   SPTP {A1 8.291, A2 -37.612, A3 70.753, A4 43.164, A5 -93.737, A6 0.000, E1 2824, E2 0, E3 0, E4 0, E5 0, E6 0} C_DIS
   SPTP {A1 8.655, A2 -38.617, A3 71.685, A4 45.116, A5 -92.691, A6 0.000, E1 2823.56, E2 0, E3 0, E4 0, E5 0, E6 0} C_DIS
   SPTP {A1 9.012, A2 -39.592, A3 72.518, A4 47.079, A5 -91.622, A6 0.000, E1 2823.06, E2 0, E3 0, E4 0, E5 0, E6 0} C_DIS
   SPTP {A1 9.360, A2 -40.537, A3 73.252, A4 49.063, A5 -90.537, A6 0.000, E1 2822.49, E2 0, E3 0, E4 0, E5 0, E6 0} C_DIS
   SPTP {A1 9.698, A2 -41.456, A3 73.903, A4 51.056, A5 -89.440, A6 0.000, E1 2821.87, E2 0, E3 0, E4 0, E5 0, E6 0} C_DIS
   SPTP {A1 10.024, A2 -42.359, A3 74.483, A4 53.057, A5 -88.326, A6 0.000, E1 2821.2, E2 0, E3 0, E4 0, E5 0, E6 0} C_DIS
   SPTP {A1 10.336, A2 -43.250, A3 75.008, A4 55.059, A5 -87.194, A6 0.000, E1 2820.49, E2 0, E3 0, E4 0, E5 0, E6 0} C_DIS
   SPTP {A1 10.632, A2 -44.132, A3 75.480, A4 57.062, A5 -86.046, A6 0.000, E1 2819.74, E2 0, E3 0, E4 0, E5 0, E6 0} C_DIS
   SPTP {A1 10.890, A2 -45.114, A3 76.113, A4 58.971, A5 -84.816, A6 0.000, E1 2818.78, E2 0, E3 0, E4 0, E5 0, E6 0} C_DIS
   SPTP {A1 11.121, A2 -46.138, A3 76.783, A4 60.845, A5 -83.533, A6 0.000, E1 2817.69, E2 0, E3 0, E4 0, E5 0, E6 0} C_DIS
   SPTP {A1 11.339, A2 -47.131, A3 77.364, A4 62.758, A5 -82.259, A6 0.000, E1 2816.52, E2 0, E3 0, E4 0, E5 0, E6 0} C_DIS
   SPTP {A1 11.539, A2 -48.119, A3 77.901, A4 64.680, A5 -80.965, A6 0.000, E1 2815.3, E2 0, E3 0, E4 0, E5 0, E6 0} C_DIS
   SPTP {A1 11.720, A2 -49.088, A3 78.371, A4 66.632, A5 -79.673, A6 0.000, E1 2814.01, E2 0, E3 0, E4 0, E5 0, E6 0} C_DIS
   SPTP {A1 11.880, A2 -50.051, A3 78.798, A4 68.601, A5 -78.370, A6 0.000, E1 2812.66, E2 0, E3 0, E4 0, E5 0, E6 0} C_DIS
   SPTP {A1 12.018, A2 -50.998, A3 79.170, A4 70.601, A5 -77.069, A6 0.000, E1 2811.24, E2 0, E3 0, E4 0, E5 0, E6 0} C_DIS
   SPTP {A1 12.134, A2 -51.928, A3 79.486, A4 72.635, A5 -75.777, A6 0.000, E1 2809.74, E2 0, E3 0, E4 0, E5 0, E6 0} C_DIS
   SPTP {A1 12.226, A2 -52.844, A3 79.754, A4 74.703, A5 -74.491, A6 0.000, E1 2808.16, E2 0, E3 0, E4 0, E5 0, E6 0} C_DIS
   SPTP {A1 12.294, A2 -53.734, A3 79.958, A4 76.821, A5 -73.233, A6 0.000, E1 2806.49, E2 0, E3 0, E4 0, E5 0, E6 0} C_DIS
   SPTP {A1 12.336, A2 -54.611, A3 80.117, A4 78.978, A5 -71.988, A6 0.000, E1 2804.74, E2 0, E3 0, E4 0, E5 0, E6 0} C_DIS
   SPTP {A1 12.353, A2 -55.450, A3 80.202, A4 81.200, A5 -70.792, A6 0.000, E1 2802.89, E2 0, E3 0, E4 0, E5 0, E6 0} C_DIS
   SPTP {A1 12.342, A2 -56.273, A3 80.242, A4 83.468, A5 -69.622, A6 0.000, E1 2800.95, E2 0, E3 0, E4 0, E5 0, E6 0} C_DIS
   SPTP {A1 12.305, A2 -57.043, A3 80.209, A4 85.765, A5 -68.529, A6 0.000, E1 2798.98, E2 0, E3 0, E4 0, E5 0, E6 0} C_DIS
   SPTP {A1 12.237, A2 -57.731, A3 80.168, A4 87.843, A5 -67.518, A6 0.000, E1 2797.48, E2 0, E3 0, E4 0, E5 0, E6 0} C_DIS
   SPTP {A1 12.145, A2 -58.394, A3 80.097, A4 89.941, A5 -66.542, A6 0.000, E1 2795.96, E2 0, E3 0, E4 0, E5 0, E6 0} C_DIS
   SPTP {A1 12.029, A2 -59.039, A3 79.995, A4 92.086, A5 -65.598, A6 0.000, E1 2794.37, E2 0, E3 0, E4 0, E5 0, E6 0} C_DIS
   SPTP {A1 11.888, A2 -59.661, A3 79.859, A4 94.281, A5 -64.695, A6 0.000, E1 2792.7, E2 0, E3 0, E4 0, E5 0, E6 0} C_DIS
   SPTP {A1 11.725, A2 -60.257, A3 79.681, A4 96.532, A5 -63.846, A6 0.000, E1 2790.95, E2 0, E3 0, E4 0, E5 0, E6 0} C_DIS
   SPTP {A1 11.538, A2 -60.826, A3 79.463, A4 98.838, A5 -63.054, A6 0.000, E1 2789.12, E2 0, E3 0, E4 0, E5 0, E6 0} C_DIS
   SPTP {A1 11.330, A2 -61.356, A3 79.191, A4 101.205, A5 -62.342, A6 0.000, E1 2787.21, E2 0, E3 0, E4 0, E5 0, E6 0} C_DIS
   SPTP {A1 11.102, A2 -61.846, A3 78.877, A4 103.596, A5 -61.710, A6 0.000, E1 2785.3, E2 0, E3 0, E4 0, E5 0, E6 0} C_DIS
   SPTP {A1 10.857, A2 -62.345, A3 78.828, A4 105.431, A5 -60.901, A6 0.000, E1 2784.47, E2 0, E3 0, E4 0, E5 0, E6 0} C_DIS
   SPTP {A1 10.594, A2 -62.833, A3 78.769, A4 107.306, A5 -60.114, A6 0.000, E1 2783.59, E2 0, E3 0, E4 0, E5 0, E6 0} C_DIS
   SPTP {A1 10.316, A2 -63.305, A3 78.697, A4 109.222, A5 -59.358, A6 0.000, E1 2782.66, E2 0, E3 0, E4 0, E5 0, E6 0} C_DIS
   SPTP {A1 10.023, A2 -63.754, A3 78.603, A4 111.183, A5 -58.650, A6 0.000, E1 2781.69, E2 0, E3 0, E4 0, E5 0, E6 0} C_DIS
   SPTP {A1 9.720, A2 -64.176, A3 78.479, A4 113.187, A5 -58.005, A6 0.000, E1 2780.67, E2 0, E3 0, E4 0, E5 0, E6 0} C_DIS
   SPTP {A1 9.408, A2 -64.567, A3 78.320, A4 115.233, A5 -57.433, A6 0.000, E1 2779.62, E2 0, E3 0, E4 0, E5 0, E6 0} C_DIS
   SPTP {A1 9.091, A2 -65.008, A3 78.418, A4 116.875, A5 -56.634, A6 0.000, E1 2779.28, E2 0, E3 0, E4 0, E5 0, E6 0} C_DIS
   SPTP {A1 8.770, A2 -65.530, A3 78.839, A4 118.046, A5 -55.511, A6 0.000, E1 2779.72, E2 0, E3 0, E4 0, E5 0, E6 0} C_DIS
   SPTP {A1 8.446, A2 -66.037, A3 79.254, A4 119.230, A5 -54.404, A6 0.000, E1 2780.16, E2 0, E3 0, E4 0, E5 0, E6 0} C_DIS
   SPTP {A1 8.121, A2 -66.525, A3 79.661, A4 120.426, A5 -53.321, A6 0.000, E1 2780.59, E2 0, E3 0, E4 0, E5 0, E6 0} C_DIS
   SPTP {A1 7.799, A2 -66.994, A3 80.058, A4 121.629, A5 -52.270, A6 0.000, E1 2781.03, E2 0, E3 0, E4 0, E5 0, E6 0} C_DIS
   SPTP {A1 7.483, A2 -67.468, A3 80.529, A4 122.693, A5 -51.156, A6 0.000, E1 2781.68, E2 0, E3 0, E4 0, E5 0, E6 0} C_DIS
   SPTP {A1 7.179, A2 -68.121, A3 81.695, A4 122.558, A5 -49.253, A6 0.000, E1 2784.01, E2 0, E3 0, E4 0, E5 0, E6 0} C_DIS
   SPTP {A1 6.881, A2 -68.742, A3 82.846, A4 122.311, A5 -47.360, A6 0.000, E1 2786.45, E2 0, E3 0, E4 0, E5 0, E6 0} C_DIS
   SPTP {A1 6.594, A2 -69.329, A3 83.978, A4 121.941, A5 -45.490, A6 0.000, E1 2788.99, E2 0, E3 0, E4 0, E5 0, E6 0} C_DIS
   SPTP {A1 6.318, A2 -69.881, A3 85.088, A4 121.431, A5 -43.647, A6 0.000, E1 2791.66, E2 0, E3 0, E4 0, E5 0, E6 0} C_DIS
   SPTP {A1 6.056, A2 -70.415, A3 86.267, A4 120.536, A5 -41.738, A6 0.000, E1 2794.76, E2 0, E3 0, E4 0, E5 0, E6 0} C_DIS
   SPTP {A1 5.815, A2 -71.014, A3 88.060, A4 117.608, A5 -39.163, A6 0.000, E1 2800.21, E2 0, E3 0, E4 0, E5 0, E6 0} C_DIS
   SPTP {A1 5.586, A2 -71.518, A3 89.769, A4 114.120, A5 -36.768, A6 0.000, E1 2806.19, E2 0, E3 0, E4 0, E5 0, E6 0} C_DIS
   SPTP {A1 5.369, A2 -71.925, A3 91.391, A4 110.015, A5 -34.596, A6 0.000, E1 2812.75, E2 0, E3 0, E4 0, E5 0, E6 0} C_DIS
   SPTP {A1 5.164, A2 -72.236, A3 92.924, A4 105.256, A5 -32.692, A6 0.000, E1 2819.92, E2 0, E3 0, E4 0, E5 0, E6 0} C_DIS
   SPTP {A1 4.973, A2 -72.448, A3 94.361, A4 99.843, A5 -31.125, A6 0.000, E1 2827.73, E2 0, E3 0, E4 0, E5 0, E6 0} C_DIS
   SPTP {A1 4.799, A2 -72.541, A3 95.781, A4 93.294, A5 -29.981, A6 0.000, E1 2836.62, E2 0, E3 0, E4 0, E5 0, E6 0} C_DIS
   SPTP {A1 4.634, A2 -72.488, A3 97.196, A4 85.489, A5 -29.420, A6 0.000, E1 2846.72, E2 0, E3 0, E4 0, E5 0, E6 0} C_DIS
   SPTP {A1 4.476, A2 -72.304, A3 98.465, A4 77.540, A5 -29.493, A6 0.000, E1 2856.93, E2 0, E3 0, E4 0, E5 0, E6 0} C_DIS
   SPTP {A1 4.325, A2 -71.991, A3 99.585, A4 69.822, A5 -30.191, A6 0.000, E1 2866.89, E2 0, E3 0, E4 0, E5 0, E6 0} C_DIS
   SPTP {A1 4.184, A2 -71.551, A3 100.551, A4 62.659, A5 -31.470, A6 0.000, E1 2876.29, E2 0, E3 0, E4 0, E5 0, E6 0} C_DIS
   SPTP {A1 4.057, A2 -70.984, A3 101.355, A4 56.273, A5 -33.255, A6 0.000, E1 2884.92, E2 0, E3 0, E4 0, E5 0, E6 0} C_DIS
   SPTP {A1 3.945, A2 -70.297, A3 101.995, A4 50.740, A5 -35.451, A6 0.000, E1 2892.7, E2 0, E3 0, E4 0, E5 0, E6 0} C_DIS
   SPTP {A1 3.847, A2 -69.498, A3 102.471, A4 46.033, A5 -37.961, A6 0.000, E1 2899.67, E2 0, E3 0, E4 0, E5 0, E6 0} C_DIS
   SPTP {A1 3.765, A2 -68.591, A3 102.779, A4 42.097, A5 -40.706, A6 0.000, E1 2905.88, E2 0, E3 0, E4 0, E5 0, E6 0} C_DIS
   SPTP {A1 3.703, A2 -67.583, A3 102.917, A4 38.849, A5 -43.620, A6 0.000, E1 2911.44, E2 0, E3 0, E4 0, E5 0, E6 0} C_DIS
   SPTP {A1 3.653, A2 -66.854, A3 102.974, A4 36.807, A5 -45.736, A6 0.000, E1 2915.49, E2 0, E3 0, E4 0, E5 0, E6 0} C_DIS
   SPTP {A1 3.624, A2 -66.078, A3 102.937, A4 35.090, A5 -47.900, A6 0.000, E1 2919.25, E2 0, E3 0, E4 0, E5 0, E6 0} C_DIS
   SPTP {A1 3.613, A2 -65.259, A3 102.808, A4 33.656, A5 -50.096, A6 0.000, E1 2922.75, E2 0, E3 0, E4 0, E5 0, E6 0} C_DIS
   SPTP {A1 3.621, A2 -64.401, A3 102.588, A4 32.476, A5 -52.305, A6 0.000, E1 2926.04, E2 0, E3 0, E4 0, E5 0, E6 0} C_DIS
   SPTP {A1 3.649, A2 -63.505, A3 102.276, A4 31.531, A5 -54.518, A6 0.000, E1 2929.12, E2 0, E3 0, E4 0, E5 0, E6 0} C_DIS
   SPTP {A1 3.697, A2 -62.577, A3 101.874, A4 30.798, A5 -56.719, A6 0.000, E1 2932.04, E2 0, E3 0, E4 0, E5 0, E6 0} C_DIS
   SPTP {A1 3.784, A2 -61.839, A3 101.495, A4 30.469, A5 -58.436, A6 0.000, E1 2934.56, E2 0, E3 0, E4 0, E5 0, E6 0} C_DIS
   SPTP {A1 3.910, A2 -61.333, A3 101.190, A4 30.506, A5 -59.622, A6 0.000, E1 2936.71, E2 0, E3 0, E4 0, E5 0, E6 0} C_DIS
   SPTP {A1 4.054, A2 -60.816, A3 100.844, A4 30.653, A5 -60.796, A6 0.000, E1 2938.79, E2 0, E3 0, E4 0, E5 0, E6 0} C_DIS
   SPTP {A1 4.213, A2 -60.292, A3 100.460, A4 30.895, A5 -61.956, A6 0.000, E1 2940.8, E2 0, E3 0, E4 0, E5 0, E6 0} C_DIS
   SPTP {A1 4.383, A2 -59.761, A3 100.041, A4 31.211, A5 -63.096, A6 0.000, E1 2942.75, E2 0, E3 0, E4 0, E5 0, E6 0} C_DIS
   SPTP {A1 4.563, A2 -59.225, A3 99.586, A4 31.603, A5 -64.215, A6 0.000, E1 2944.66, E2 0, E3 0, E4 0, E5 0, E6 0} C_DIS
   SPTP {A1 4.753, A2 -58.683, A3 99.094, A4 32.066, A5 -65.312, A6 0.000, E1 2946.51, E2 0, E3 0, E4 0, E5 0, E6 0} C_DIS
   SPTP {A1 4.951, A2 -58.137, A3 98.569, A4 32.587, A5 -66.385, A6 0.000, E1 2948.32, E2 0, E3 0, E4 0, E5 0, E6 0} C_DIS
   SPTP {A1 5.200, A2 -57.839, A3 98.169, A4 33.422, A5 -66.957, A6 0.000, E1 2949.88, E2 0, E3 0, E4 0, E5 0, E6 0} C_DIS
   SPTP {A1 5.478, A2 -57.668, A3 97.826, A4 34.439, A5 -67.271, A6 0.000, E1 2951.28, E2 0, E3 0, E4 0, E5 0, E6 0} C_DIS
   SPTP {A1 5.759, A2 -57.494, A3 97.460, A4 35.497, A5 -67.574, A6 0.000, E1 2952.65, E2 0, E3 0, E4 0, E5 0, E6 0} C_DIS
   SPTP {A1 6.043, A2 -57.319, A3 97.070, A4 36.589, A5 -67.865, A6 0.000, E1 2953.99, E2 0, E3 0, E4 0, E5 0, E6 0} C_DIS
   SPTP {A1 6.327, A2 -57.140, A3 96.658, A4 37.712, A5 -68.146, A6 0.000, E1 2955.29, E2 0, E3 0, E4 0, E5 0, E6 0} C_DIS
   SPTP {A1 6.613, A2 -56.959, A3 96.222, A4 38.865, A5 -68.416, A6 0.000, E1 2956.57, E2 0, E3 0, E4 0, E5 0, E6 0} C_DIS
   SPTP {A1 6.896, A2 -56.775, A3 95.765, A4 40.039, A5 -68.676, A6 0.000, E1 2957.82, E2 0, E3 0, E4 0, E5 0, E6 0} C_DIS
   SPTP {A1 7.178, A2 -56.589, A3 95.287, A4 41.232, A5 -68.926, A6 0.000, E1 2959.05, E2 0, E3 0, E4 0, E5 0, E6 0} C_DIS
   SPTP {A1 7.456, A2 -56.402, A3 94.790, A4 42.440, A5 -69.166, A6 0.000, E1 2960.26, E2 0, E3 0, E4 0, E5 0, E6 0} C_DIS
   SPTP {A1 7.729, A2 -56.213, A3 94.273, A4 43.658, A5 -69.394, A6 0.000, E1 2961.45, E2 0, E3 0, E4 0, E5 0, E6 0} C_DIS
   SPTP {A1 7.996, A2 -56.024, A3 93.742, A4 44.880, A5 -69.610, A6 0.000, E1 2962.63, E2 0, E3 0, E4 0, E5 0, E6 0} C_DIS
   SPTP {A1 8.257, A2 -55.836, A3 93.196, A4 46.105, A5 -69.815, A6 0.000, E1 2963.81, E2 0, E3 0, E4 0, E5 0, E6 0} C_DIS
   SPTP {A1 8.523, A2 -55.760, A3 92.717, A4 47.443, A5 -69.822, A6 0.000, E1 2964.79, E2 0, E3 0, E4 0, E5 0, E6 0} C_DIS
   SPTP {A1 8.783, A2 -55.694, A3 92.230, A4 48.797, A5 -69.805, A6 0.000, E1 2965.75, E2 0, E3 0, E4 0, E5 0, E6 0} C_DIS
   SPTP {A1 9.034, A2 -55.626, A3 91.728, A4 50.152, A5 -69.783, A6 0.000, E1 2966.69, E2 0, E3 0, E4 0, E5 0, E6 0} C_DIS
   SPTP {A1 9.278, A2 -55.557, A3 91.213, A4 51.506, A5 -69.757, A6 0.000, E1 2967.63, E2 0, E3 0, E4 0, E5 0, E6 0} C_DIS
   SPTP {A1 9.512, A2 -55.488, A3 90.688, A4 52.857, A5 -69.725, A6 0.000, E1 2968.55, E2 0, E3 0, E4 0, E5 0, E6 0} C_DIS
   SPTP {A1 9.737, A2 -55.420, A3 90.153, A4 54.202, A5 -69.688, A6 0.000, E1 2969.47, E2 0, E3 0, E4 0, E5 0, E6 0} C_DIS
   SPTP {A1 9.953, A2 -55.353, A3 89.611, A4 55.538, A5 -69.645, A6 0.000, E1 2970.39, E2 0, E3 0, E4 0, E5 0, E6 0} C_DIS
   SPTP {A1 10.158, A2 -55.289, A3 89.065, A4 56.865, A5 -69.594, A6 0.000, E1 2971.3, E2 0, E3 0, E4 0, E5 0, E6 0} C_DIS
   SPTP {A1 10.352, A2 -55.227, A3 88.515, A4 58.180, A5 -69.536, A6 0.000, E1 2972.22, E2 0, E3 0, E4 0, E5 0, E6 0} C_DIS
   SPTP {A1 10.536, A2 -55.171, A3 87.966, A4 59.481, A5 -69.468, A6 0.000, E1 2973.14, E2 0, E3 0, E4 0, E5 0, E6 0} C_DIS
   SPTP {A1 10.700, A2 -55.122, A3 87.442, A4 60.719, A5 -69.407, A6 0.000, E1 2974.04, E2 0, E3 0, E4 0, E5 0, E6 0} C_DIS
   SPTP {A1 10.850, A2 -55.080, A3 86.931, A4 61.923, A5 -69.341, A6 0.000, E1 2974.94, E2 0, E3 0, E4 0, E5 0, E6 0} C_DIS
   SPTP {A1 10.965, A2 -55.046, A3 86.490, A4 62.972, A5 -69.312, A6 0.000, E1 2975.8, E2 0, E3 0, E4 0, E5 0, E6 0} C_DIS
   SPTP {A1 11.068, A2 -55.022, A3 86.067, A4 63.988, A5 -69.273, A6 0.000, E1 2976.66, E2 0, E3 0, E4 0, E5 0, E6 0} C_DIS
   SPTP {A1 11.164, A2 -55.008, A3 85.655, A4 64.986, A5 -69.221, A6 0.000, E1 2977.54, E2 0, E3 0, E4 0, E5 0, E6 0} C_DIS
   SPTP {A1 11.250, A2 -55.004, A3 85.258, A4 65.965, A5 -69.153, A6 0.000, E1 2978.43, E2 0, E3 0, E4 0, E5 0, E6 0} C_DIS
   SPTP {A1 11.329, A2 -55.012, A3 84.876, A4 66.925, A5 -69.067, A6 0.000, E1 2979.34, E2 0, E3 0, E4 0, E5 0, E6 0} C_DIS
   SPTP {A1 11.400, A2 -55.031, A3 84.511, A4 67.865, A5 -68.964, A6 0.000, E1 2980.26, E2 0, E3 0, E4 0, E5 0, E6 0} C_DIS
   SPTP {A1 11.462, A2 -55.065, A3 84.166, A4 68.784, A5 -68.840, A6 0.000, E1 2981.19, E2 0, E3 0, E4 0, E5 0, E6 0} C_DIS
   SPTP {A1 11.516, A2 -55.112, A3 83.842, A4 69.683, A5 -68.696, A6 0.000, E1 2982.14, E2 0, E3 0, E4 0, E5 0, E6 0} C_DIS
   SPTP {A1 11.562, A2 -55.174, A3 83.539, A4 70.561, A5 -68.529, A6 0.000, E1 2983.1, E2 0, E3 0, E4 0, E5 0, E6 0} C_DIS
   SPTP {A1 11.600, A2 -55.251, A3 83.260, A4 71.418, A5 -68.340, A6 0.000, E1 2984.08, E2 0, E3 0, E4 0, E5 0, E6 0} C_DIS
   SPTP {A1 11.630, A2 -55.344, A3 83.006, A4 72.254, A5 -68.126, A6 0.000, E1 2985.08, E2 0, E3 0, E4 0, E5 0, E6 0} C_DIS
   SPTP {A1 11.652, A2 -55.453, A3 82.777, A4 73.069, A5 -67.888, A6 0.000, E1 2986.09, E2 0, E3 0, E4 0, E5 0, E6 0} C_DIS
   SPTP {A1 11.666, A2 -55.579, A3 82.575, A4 73.863, A5 -67.625, A6 0.000, E1 2987.12, E2 0, E3 0, E4 0, E5 0, E6 0} C_DIS
   SPTP {A1 11.672, A2 -55.721, A3 82.401, A4 74.635, A5 -67.334, A6 0.000, E1 2988.17, E2 0, E3 0, E4 0, E5 0, E6 0} C_DIS
   SPTP {A1 11.671, A2 -55.881, A3 82.255, A4 75.387, A5 -67.016, A6 0.000, E1 2989.23, E2 0, E3 0, E4 0, E5 0, E6 0} C_DIS
   SPTP {A1 11.661, A2 -56.058, A3 82.138, A4 76.117, A5 -66.670, A6 0.000, E1 2990.3, E2 0, E3 0, E4 0, E5 0, E6 0} C_DIS
   SPTP {A1 11.644, A2 -56.253, A3 82.050, A4 76.826, A5 -66.293, A6 0.000, E1 2991.4, E2 0, E3 0, E4 0, E5 0, E6 0} C_DIS
   SPTP {A1 11.611, A2 -56.512, A3 82.046, A4 77.547, A5 -65.858, A6 0.000, E1 2992.22, E2 0, E3 0, E4 0, E5 0, E6 0} C_DIS
   SPTP {A1 11.571, A2 -56.791, A3 82.070, A4 78.258, A5 -65.397, A6 0.000, E1 2993.02, E2 0, E3 0, E4 0, E5 0, E6 0} C_DIS
   SPTP {A1 11.523, A2 -57.080, A3 82.113, A4 78.957, A5 -64.914, A6 0.000, E1 2993.82, E2 0, E3 0, E4 0, E5 0, E6 0} C_DIS
   SPTP {A1 11.468, A2 -57.383, A3 82.178, A4 79.641, A5 -64.406, A6 0.000, E1 2994.62, E2 0, E3 0, E4 0, E5 0, E6 0} C_DIS
   SPTP {A1 11.406, A2 -57.697, A3 82.264, A4 80.312, A5 -63.873, A6 0.000, E1 2995.44, E2 0, E3 0, E4 0, E5 0, E6 0} C_DIS
   SPTP {A1 11.336, A2 -58.025, A3 82.371, A4 80.968, A5 -63.314, A6 0.000, E1 2996.26, E2 0, E3 0, E4 0, E5 0, E6 0} C_DIS
   SPTP {A1 11.258, A2 -58.365, A3 82.500, A4 81.609, A5 -62.728, A6 0.000, E1 2997.08, E2 0, E3 0, E4 0, E5 0, E6 0} C_DIS
   SPTP {A1 11.173, A2 -58.718, A3 82.651, A4 82.236, A5 -62.114, A6 0.000, E1 2997.91, E2 0, E3 0, E4 0, E5 0, E6 0} C_DIS
   SPTP {A1 11.079, A2 -59.083, A3 82.823, A4 82.849, A5 -61.473, A6 0.000, E1 2998.75, E2 0, E3 0, E4 0, E5 0, E6 0} C_DIS
   SPTP {A1 10.977, A2 -59.459, A3 83.015, A4 83.448, A5 -60.804, A6 0.000, E1 2999.59, E2 0, E3 0, E4 0, E5 0, E6 0} C_DIS
   SPTP {A1 10.867, A2 -59.846, A3 83.228, A4 84.033, A5 -60.106, A6 0.000, E1 3000.43, E2 0, E3 0, E4 0, E5 0, E6 0} C_DIS
   SPTP {A1 10.748, A2 -60.245, A3 83.460, A4 84.605, A5 -59.379, A6 0.000, E1 3001.28, E2 0, E3 0, E4 0, E5 0, E6 0} C_DIS
   SPTP {A1 10.629, A2 -60.717, A3 83.597, A4 85.698, A5 -58.495, A6 0.000, E1 3001.52, E2 0, E3 0, E4 0, E5 0, E6 0} C_DIS
   SPTP {A1 10.498, A2 -61.191, A3 83.738, A4 86.804, A5 -57.596, A6 0.000, E1 3001.74, E2 0, E3 0, E4 0, E5 0, E6 0} C_DIS
   SPTP {A1 10.355, A2 -61.668, A3 83.884, A4 87.922, A5 -56.684, A6 0.000, E1 3001.94, E2 0, E3 0, E4 0, E5 0, E6 0} C_DIS
   SPTP {A1 10.201, A2 -62.146, A3 84.036, A4 89.054, A5 -55.758, A6 0.000, E1 3002.1, E2 0, E3 0, E4 0, E5 0, E6 0} C_DIS
   SPTP {A1 10.036, A2 -62.624, A3 84.192, A4 90.203, A5 -54.820, A6 0.000, E1 3002.24, E2 0, E3 0, E4 0, E5 0, E6 0} C_DIS
   SPTP {A1 9.859, A2 -63.102, A3 84.351, A4 91.371, A5 -53.873, A6 0.000, E1 3002.35, E2 0, E3 0, E4 0, E5 0, E6 0} C_DIS
   SPTP {A1 9.670, A2 -63.579, A3 84.513, A4 92.559, A5 -52.914, A6 0.000, E1 3002.42, E2 0, E3 0, E4 0, E5 0, E6 0} C_DIS
   SPTP {A1 9.469, A2 -64.055, A3 84.678, A4 93.770, A5 -51.944, A6 0.000, E1 3002.46, E2 0, E3 0, E4 0, E5 0, E6 0} C_DIS
   SPTP {A1 9.257, A2 -64.531, A3 84.846, A4 95.006, A5 -50.964, A6 0.000, E1 3002.46, E2 0, E3 0, E4 0, E5 0, E6 0} C_DIS
   SPTP {A1 9.032, A2 -65.004, A3 85.017, A4 96.271, A5 -49.974, A6 0.000, E1 3002.43, E2 0, E3 0, E4 0, E5 0, E6 0} C_DIS
   SPTP {A1 8.795, A2 -65.475, A3 85.190, A4 97.566, A5 -48.977, A6 0.000, E1 3002.34, E2 0, E3 0, E4 0, E5 0, E6 0} C_DIS
   SPTP {A1 8.545, A2 -65.943, A3 85.363, A4 98.896, A5 -47.972, A6 0.000, E1 3002.22, E2 0, E3 0, E4 0, E5 0, E6 0} C_DIS
   SPTP {A1 8.284, A2 -66.407, A3 85.538, A4 100.264, A5 -46.962, A6 0.000, E1 3002.04, E2 0, E3 0, E4 0, E5 0, E6 0} C_DIS
   SPTP {A1 8.011, A2 -66.866, A3 85.711, A4 101.674, A5 -45.950, A6 0.000, E1 3001.81, E2 0, E3 0, E4 0, E5 0, E6 0} C_DIS
   SPTP {A1 7.724, A2 -67.320, A3 85.859, A4 103.228, A5 -44.926, A6 0.000, E1 3001.47, E2 0, E3 0, E4 0, E5 0, E6 0} C_DIS
   SPTP {A1 7.411, A2 -67.777, A3 85.920, A4 105.216, A5 -43.841, A6 0.000, E1 3000.88, E2 0, E3 0, E4 0, E5 0, E6 0} C_DIS
   SPTP {A1 7.084, A2 -68.223, A3 85.976, A4 107.281, A5 -42.777, A6 0.000, E1 3000.19, E2 0, E3 0, E4 0, E5 0, E6 0} C_DIS
   SPTP {A1 6.742, A2 -68.658, A3 86.030, A4 109.428, A5 -41.733, A6 0.000, E1 2999.42, E2 0, E3 0, E4 0, E5 0, E6 0} C_DIS
   SPTP {A1 6.386, A2 -69.081, A3 86.080, A4 111.660, A5 -40.713, A6 0.000, E1 2998.55, E2 0, E3 0, E4 0, E5 0, E6 0} C_DIS
   SPTP {A1 6.016, A2 -69.492, A3 86.128, A4 113.983, A5 -39.720, A6 0.000, E1 2997.59, E2 0, E3 0, E4 0, E5 0, E6 0} C_DIS
   SPTP {A1 5.634, A2 -69.889, A3 86.169, A4 116.400, A5 -38.763, A6 0.000, E1 2996.52, E2 0, E3 0, E4 0, E5 0, E6 0} C_DIS
   SPTP {A1 5.240, A2 -70.272, A3 86.205, A4 118.913, A5 -37.851, A6 0.000, E1 2995.36, E2 0, E3 0, E4 0, E5 0, E6 0} C_DIS
   SPTP {A1 4.837, A2 -70.638, A3 86.234, A4 121.523, A5 -36.988, A6 0.000, E1 2994.11, E2 0, E3 0, E4 0, E5 0, E6 0} C_DIS
   SPTP {A1 4.425, A2 -70.989, A3 86.256, A4 124.227, A5 -36.181, A6 0.000, E1 2992.76, E2 0, E3 0, E4 0, E5 0, E6 0} C_DIS
   SPTP {A1 4.006, A2 -71.322, A3 86.271, A4 127.019, A5 -35.437, A6 0.000, E1 2991.32, E2 0, E3 0, E4 0, E5 0, E6 0} C_DIS
   SPTP {A1 3.581, A2 -71.639, A3 86.281, A4 129.897, A5 -34.756, A6 0.000, E1 2989.81, E2 0, E3 0, E4 0, E5 0, E6 0} C_DIS
   SPTP {A1 3.149, A2 -71.941, A3 86.286, A4 132.852, A5 -34.141, A6 0.000, E1 2988.23, E2 0, E3 0, E4 0, E5 0, E6 0} C_DIS
   SPTP {A1 2.715, A2 -72.225, A3 86.284, A4 135.865, A5 -33.605, A6 0.000, E1 2986.6, E2 0, E3 0, E4 0, E5 0, E6 0} C_DIS
   SPTP {A1 2.281, A2 -72.555, A3 86.514, A4 138.429, A5 -32.773, A6 0.000, E1 2985.54, E2 0, E3 0, E4 0, E5 0, E6 0} C_DIS
   SPTP {A1 1.845, A2 -72.929, A3 86.959, A4 140.623, A5 -31.635, A6 0.000, E1 2984.96, E2 0, E3 0, E4 0, E5 0, E6 0} C_DIS
   SPTP {A1 1.413, A2 -73.291, A3 87.411, A4 142.897, A5 -30.522, A6 0.000, E1 2984.3, E2 0, E3 0, E4 0, E5 0, E6 0} C_DIS
   SPTP {A1 0.983, A2 -73.642, A3 87.869, A4 145.255, A5 -29.433, A6 0.000, E1 2983.56, E2 0, E3 0, E4 0, E5 0, E6 0} C_DIS
   SPTP {A1 0.564, A2 -73.981, A3 88.333, A4 147.674, A5 -28.380, A6 0.000, E1 2982.77, E2 0, E3 0, E4 0, E5 0, E6 0} C_DIS
   SPTP {A1 0.158, A2 -74.307, A3 88.803, A4 150.140, A5 -27.366, A6 0.000, E1 2981.96, E2 0, E3 0, E4 0, E5 0, E6 0} C_DIS
   SPTP {A1 -0.229, A2 -74.622, A3 89.278, A4 152.627, A5 -26.396, A6 0.000, E1 2981.14, E2 0, E3 0, E4 0, E5 0, E6 0} C_DIS
   SPTP {A1 -0.592, A2 -74.973, A3 89.961, A4 154.675, A5 -25.088, A6 0.000, E1 2980.8, E2 0, E3 0, E4 0, E5 0, E6 0} C_DIS
   SPTP {A1 -0.921, A2 -75.415, A3 91.154, A4 155.531, A5 -22.825, A6 0.000, E1 2981.64, E2 0, E3 0, E4 0, E5 0, E6 0} C_DIS
   SPTP {A1 -1.221, A2 -75.822, A3 92.330, A4 156.269, A5 -20.565, A6 0.000, E1 2982.62, E2 0, E3 0, E4 0, E5 0, E6 0} C_DIS
   SPTP {A1 -1.484, A2 -76.194, A3 93.486, A4 156.798, A5 -18.315, A6 0.000, E1 2983.83, E2 0, E3 0, E4 0, E5 0, E6 0} C_DIS
   SPTP {A1 -1.707, A2 -76.530, A3 94.623, A4 156.983, A5 -16.077, A6 0.000, E1 2985.4, E2 0, E3 0, E4 0, E5 0, E6 0} C_DIS
   SPTP {A1 -1.878, A2 -76.847, A3 95.938, A4 155.655, A5 -13.412, A6 0.000, E1 2988.51, E2 0, E3 0, E4 0, E5 0, E6 0} C_DIS
   SPTP {A1 -2.003, A2 -77.121, A3 97.769, A4 148.572, A5 -9.513, A6 0.000, E1 2997.32, E2 0, E3 0, E4 0, E5 0, E6 0} C_DIS
   SPTP {A1 -2.073, A2 -77.268, A3 99.483, A4 131.076, A5 -6.066, A6 0.000, E1 3016.55, E2 0, E3 0, E4 0, E5 0, E6 0} C_DIS
   SPTP {A1 -2.095, A2 -77.287, A3 101.076, A4 87.723, A5 -4.353, A6 0.000, E1 3061.65, E2 0, E3 0, E4 0, E5 0, E6 0} C_DIS
   SPTP {A1 -2.058, A2 -77.175, A3 102.538, A4 44.883, A5 -6.134, A6 0.000, E1 3106.26, E2 0, E3 0, E4 0, E5 0, E6 0} C_DIS
   SPTP {A1 -1.985, A2 -76.714, A3 104.288, A4 23.426, A5 -11.222, A6 0.000, E1 3129.5, E2 0, E3 0, E4 0, E5 0, E6 0} C_DIS
   SPTP {A1 -1.870, A2 -75.910, A3 105.843, A4 15.959, A5 -17.402, A6 0.000, E1 3138.75, E2 0, E3 0, E4 0, E5 0, E6 0} C_DIS
   SPTP {A1 -1.718, A2 -74.815, A3 107.046, A4 12.881, A5 -23.708, A6 0.000, E1 3143.62, E2 0, E3 0, E4 0, E5 0, E6 0} C_DIS
   SPTP {A1 -1.548, A2 -73.241, A3 107.939, A4 11.064, A5 -30.738, A6 0.000, E1 3147.32, E2 0, E3 0, E4 0, E5 0, E6 0} C_DIS
   SPTP {A1 -1.356, A2 -70.901, A3 108.348, A4 9.830, A5 -39.024, A6 0.000, E1 3150.66, E2 0, E3 0, E4 0, E5 0, E6 0} C_DIS
   SPTP {A1 -1.158, A2 -68.174, A3 108.071, A4 9.263, A5 -47.048, A6 0.000, E1 3153.34, E2 0, E3 0, E4 0, E5 0, E6 0} C_DIS
   SPTP {A1 -0.962, A2 -65.135, A3 107.107, A4 9.065, A5 -54.717, A6 0.000, E1 3155.68, E2 0, E3 0, E4 0, E5 0, E6 0} C_DIS
   SPTP {A1 -0.727, A2 -62.038, A3 105.570, A4 9.217, A5 -61.595, A6 0.000, E1 3157.91, E2 0, E3 0, E4 0, E5 0, E6 0} C_DIS
   SPTP {A1 -0.305, A2 -59.408, A3 103.857, A4 10.064, A5 -66.874, A6 0.000, E1 3160.23, E2 0, E3 0, E4 0, E5 0, E6 0} C_DIS
   SPTP {A1 0.131, A2 -56.724, A3 101.755, A4 11.050, A5 -71.795, A6 0.000, E1 3162.51, E2 0, E3 0, E4 0, E5 0, E6 0} C_DIS
   SPTP {A1 0.584, A2 -54.011, A3 99.275, A4 12.190, A5 -76.346, A6 0.000, E1 3164.75, E2 0, E3 0, E4 0, E5 0, E6 0} C_DIS
   SPTP {A1 1.046, A2 -51.291, A3 96.439, A4 13.453, A5 -80.520, A6 0.000, E1 3166.97, E2 0, E3 0, E4 0, E5 0, E6 0} C_DIS
   SPTP {A1 1.511, A2 -48.578, A3 93.262, A4 14.831, A5 -84.315, A6 0.000, E1 3169.17, E2 0, E3 0, E4 0, E5 0, E6 0} C_DIS
   SPTP {A1 1.980, A2 -45.874, A3 89.752, A4 16.327, A5 -87.740, A6 0.000, E1 3171.33, E2 0, E3 0, E4 0, E5 0, E6 0} C_DIS
   SPTP {A1 2.453, A2 -43.174, A3 85.904, A4 17.952, A5 -90.804, A6 0.000, E1 3173.44, E2 0, E3 0, E4 0, E5 0, E6 0} C_DIS
   SPTP {A1 2.923, A2 -40.469, A3 81.717, A4 19.679, A5 -93.514, A6 0.000, E1 3175.49, E2 0, E3 0, E4 0, E5 0, E6 0} C_DIS
   SPTP {A1 3.388, A2 -37.736, A3 77.160, A4 21.509, A5 -95.879, A6 0.000, E1 3177.44, E2 0, E3 0, E4 0, E5 0, E6 0} C_DIS
   SPTP {A1 3.843, A2 -34.945, A3 72.200, A4 23.417, A5 -97.903, A6 0.000, E1 3179.27, E2 0, E3 0, E4 0, E5 0, E6 0} C_DIS
   SPTP {A1 4.407, A2 -34.766, A3 71.380, A4 25.593, A5 -97.876, A6 0.000, E1 3180.54, E2 0, E3 0, E4 0, E5 0, E6 0} C_DIS
   SPTP {A1 4.967, A2 -34.634, A3 70.580, A4 27.841, A5 -97.769, A6 0.000, E1 3181.65, E2 0, E3 0, E4 0, E5 0, E6 0} C_DIS
   SPTP {A1 5.517, A2 -34.477, A3 69.685, A4 30.139, A5 -97.636, A6 0.000, E1 3182.61, E2 0, E3 0, E4 0, E5 0, E6 0} C_DIS
   SPTP {A1 6.038, A2 -34.559, A3 69.172, A4 32.400, A5 -97.327, A6 0.000, E1 3183.34, E2 0, E3 0, E4 0, E5 0, E6 0} C_DIS
   SPTP {A1 6.516, A2 -35.196, A3 69.605, A4 34.539, A5 -96.655, A6 0.000, E1 3183.71, E2 0, E3 0, E4 0, E5 0, E6 0} C_DIS
   SPTP {A1 6.983, A2 -35.782, A3 69.912, A4 36.702, A5 -95.978, A6 0.000, E1 3183.95, E2 0, E3 0, E4 0, E5 0, E6 0} C_DIS
   SPTP {A1 7.440, A2 -36.329, A3 70.111, A4 38.888, A5 -95.294, A6 0.000, E1 3184.09, E2 0, E3 0, E4 0, E5 0, E6 0} C_DIS
   SPTP {A1 7.441, A2 -36.315, A3 70.093, A4 38.902, A5 -95.305, A6 0.000, E1 3184.07, E2 0, E3 0, E4 0, E5 0, E6 0} C_DIS
   SPTP {A1 7.888, A2 -36.831, A3 70.201, A4 41.107, A5 -94.614, A6 0.000, E1 3184.15, E2 0, E3 0, E4 0, E5 0, E6 0} C_DIS
   SPTP {A1 8.292, A2 -37.590, A3 70.724, A4 43.181, A5 -93.755, A6 0.000, E1 3183.98, E2 0, E3 0, E4 0, E5 0, E6 0} C_DIS
   SPTP {A1 8.656, A2 -38.593, A3 71.652, A4 45.135, A5 -92.711, A6 0.000, E1 3183.53, E2 0, E3 0, E4 0, E5 0, E6 0} C_DIS
   SPTP {A1 9.013, A2 -39.567, A3 72.483, A4 47.099, A5 -91.644, A6 0.000, E1 3183.03, E2 0, E3 0, E4 0, E5 0, E6 0} C_DIS
   SPTP {A1 9.362, A2 -40.510, A3 73.216, A4 49.084, A5 -90.562, A6 0.000, E1 3182.46, E2 0, E3 0, E4 0, E5 0, E6 0} C_DIS
   SPTP {A1 9.700, A2 -41.428, A3 73.864, A4 51.078, A5 -89.467, A6 0.000, E1 3181.83, E2 0, E3 0, E4 0, E5 0, E6 0} C_DIS
   SPTP {A1 10.026, A2 -42.329, A3 74.443, A4 53.080, A5 -88.355, A6 0.000, E1 3181.17, E2 0, E3 0, E4 0, E5 0, E6 0} C_DIS
   SPTP {A1 10.338, A2 -43.220, A3 74.967, A4 55.082, A5 -87.225, A6 0.000, E1 3180.46, E2 0, E3 0, E4 0, E5 0, E6 0} C_DIS
   SPTP {A1 10.634, A2 -44.100, A3 75.438, A4 57.085, A5 -86.079, A6 0.000, E1 3179.71, E2 0, E3 0, E4 0, E5 0, E6 0} C_DIS
   SPTP {A1 10.892, A2 -45.082, A3 76.070, A4 58.995, A5 -84.852, A6 0.000, E1 3178.75, E2 0, E3 0, E4 0, E5 0, E6 0} C_DIS
   SPTP {A1 11.124, A2 -46.105, A3 76.740, A4 60.870, A5 -83.571, A6 0.000, E1 3177.66, E2 0, E3 0, E4 0, E5 0, E6 0} C_DIS
   SPTP {A1 11.342, A2 -47.097, A3 77.320, A4 62.782, A5 -82.299, A6 0.000, E1 3176.49, E2 0, E3 0, E4 0, E5 0, E6 0} C_DIS
   SPTP {A1 11.542, A2 -48.085, A3 77.857, A4 64.705, A5 -81.006, A6 0.000, E1 3175.27, E2 0, E3 0, E4 0, E5 0, E6 0} C_DIS
   SPTP {A1 11.723, A2 -49.054, A3 78.327, A4 66.656, A5 -79.716, A6 0.000, E1 3173.98, E2 0, E3 0, E4 0, E5 0, E6 0} C_DIS
   SPTP {A1 11.883, A2 -50.016, A3 78.755, A4 68.625, A5 -78.414, A6 0.000, E1 3172.64, E2 0, E3 0, E4 0, E5 0, E6 0} C_DIS
   SPTP {A1 12.022, A2 -50.963, A3 79.127, A4 70.624, A5 -77.116, A6 0.000, E1 3171.21, E2 0, E3 0, E4 0, E5 0, E6 0} C_DIS
   SPTP {A1 12.139, A2 -51.893, A3 79.444, A4 72.657, A5 -75.825, A6 0.000, E1 3169.72, E2 0, E3 0, E4 0, E5 0, E6 0} C_DIS
   SPTP {A1 12.231, A2 -52.810, A3 79.713, A4 74.725, A5 -74.540, A6 0.000, E1 3168.14, E2 0, E3 0, E4 0, E5 0, E6 0} C_DIS
   SPTP {A1 12.299, A2 -53.700, A3 79.917, A4 76.841, A5 -73.283, A6 0.000, E1 3166.48, E2 0, E3 0, E4 0, E5 0, E6 0} C_DIS
   SPTP {A1 12.341, A2 -54.576, A3 80.078, A4 78.997, A5 -72.039, A6 0.000, E1 3164.73, E2 0, E3 0, E4 0, E5 0, E6 0} C_DIS
   SPTP {A1 12.359, A2 -55.416, A3 80.163, A4 81.217, A5 -70.844, A6 0.000, E1 3162.88, E2 0, E3 0, E4 0, E5 0, E6 0} C_DIS
   SPTP {A1 12.348, A2 -56.240, A3 80.205, A4 83.484, A5 -69.674, A6 0.000, E1 3160.94, E2 0, E3 0, E4 0, E5 0, E6 0} C_DIS
   SPTP {A1 12.311, A2 -57.011, A3 80.174, A4 85.778, A5 -68.581, A6 0.000, E1 3158.98, E2 0, E3 0, E4 0, E5 0, E6 0} C_DIS
   SPTP {A1 12.243, A2 -57.699, A3 80.134, A4 87.855, A5 -67.569, A6 0.000, E1 3157.48, E2 0, E3 0, E4 0, E5 0, E6 0} C_DIS
   SPTP {A1 12.152, A2 -58.363, A3 80.065, A4 89.951, A5 -66.593, A6 0.000, E1 3155.96, E2 0, E3 0, E4 0, E5 0, E6 0} C_DIS
   SPTP {A1 12.036, A2 -59.009, A3 79.965, A4 92.092, A5 -65.648, A6 0.000, E1 3154.38, E2 0, E3 0, E4 0, E5 0, E6 0} C_DIS
   SPTP {A1 11.896, A2 -59.633, A3 79.830, A4 94.285, A5 -64.745, A6 0.000, E1 3152.71, E2 0, E3 0, E4 0, E5 0, E6 0} C_DIS
   SPTP {A1 11.732, A2 -60.230, A3 79.655, A4 96.533, A5 -63.895, A6 0.000, E1 3150.96, E2 0, E3 0, E4 0, E5 0, E6 0} C_DIS
   SPTP {A1 11.545, A2 -60.799, A3 79.440, A4 98.835, A5 -63.101, A6 0.000, E1 3149.14, E2 0, E3 0, E4 0, E5 0, E6 0} C_DIS
   SPTP {A1 11.337, A2 -61.331, A3 79.170, A4 101.199, A5 -62.386, A6 0.000, E1 3147.23, E2 0, E3 0, E4 0, E5 0, E6 0} C_DIS
   SPTP {A1 11.110, A2 -61.823, A3 78.857, A4 103.591, A5 -61.753, A6 0.000, E1 3145.31, E2 0, E3 0, E4 0, E5 0, E6 0} C_DIS
   SPTP {A1 10.864, A2 -62.323, A3 78.810, A4 105.423, A5 -60.942, A6 0.000, E1 3144.49, E2 0, E3 0, E4 0, E5 0, E6 0} C_DIS
   SPTP {A1 10.602, A2 -62.812, A3 78.754, A4 107.295, A5 -60.152, A6 0.000, E1 3143.61, E2 0, E3 0, E4 0, E5 0, E6 0} C_DIS
   SPTP {A1 10.323, A2 -63.286, A3 78.685, A4 109.208, A5 -59.393, A6 0.000, E1 3142.69, E2 0, E3 0, E4 0, E5 0, E6 0} C_DIS
   SPTP {A1 10.031, A2 -63.737, A3 78.593, A4 111.166, A5 -58.682, A6 0.000, E1 3141.71, E2 0, E3 0, E4 0, E5 0, E6 0} C_DIS
   SPTP {A1 9.728, A2 -64.161, A3 78.471, A4 113.167, A5 -58.034, A6 0.000, E1 3140.7, E2 0, E3 0, E4 0, E5 0, E6 0} C_DIS
   SPTP {A1 9.416, A2 -64.553, A3 78.315, A4 115.210, A5 -57.458, A6 0.000, E1 3139.65, E2 0, E3 0, E4 0, E5 0, E6 0} C_DIS
   SPTP {A1 9.098, A2 -64.995, A3 78.410, A4 116.859, A5 -56.662, A6 0.000, E1 3139.29, E2 0, E3 0, E4 0, E5 0, E6 0} C_DIS
   SPTP {A1 8.776, A2 -65.518, A3 78.833, A4 118.029, A5 -55.534, A6 0.000, E1 3139.73, E2 0, E3 0, E4 0, E5 0, E6 0} C_DIS
   SPTP {A1 8.452, A2 -66.026, A3 79.251, A4 119.211, A5 -54.423, A6 0.000, E1 3140.17, E2 0, E3 0, E4 0, E5 0, E6 0} C_DIS
   SPTP {A1 8.126, A2 -66.517, A3 79.661, A4 120.405, A5 -53.336, A6 0.000, E1 3140.6, E2 0, E3 0, E4 0, E5 0, E6 0} C_DIS
   SPTP {A1 7.804, A2 -66.987, A3 80.059, A4 121.607, A5 -52.282, A6 0.000, E1 3141.03, E2 0, E3 0, E4 0, E5 0, E6 0} C_DIS
   SPTP {A1 7.487, A2 -67.459, A3 80.522, A4 122.689, A5 -51.177, A6 0.000, E1 3141.65, E2 0, E3 0, E4 0, E5 0, E6 0} C_DIS
   SPTP {A1 7.182, A2 -68.113, A3 81.688, A4 122.555, A5 -49.272, A6 0.000, E1 3143.98, E2 0, E3 0, E4 0, E5 0, E6 0} C_DIS
   SPTP {A1 6.884, A2 -68.736, A3 82.840, A4 122.312, A5 -47.376, A6 0.000, E1 3146.41, E2 0, E3 0, E4 0, E5 0, E6 0} C_DIS
   SPTP {A1 6.595, A2 -69.324, A3 83.972, A4 121.944, A5 -45.503, A6 0.000, E1 3148.94, E2 0, E3 0, E4 0, E5 0, E6 0} C_DIS
   SPTP {A1 6.318, A2 -69.877, A3 85.083, A4 121.439, A5 -43.658, A6 0.000, E1 3151.61, E2 0, E3 0, E4 0, E5 0, E6 0} C_DIS
   SPTP {A1 6.055, A2 -70.409, A3 86.248, A4 120.584, A5 -41.762, A6 0.000, E1 3154.65, E2 0, E3 0, E4 0, E5 0, E6 0} C_DIS
   SPTP {A1 5.812, A2 -71.010, A3 88.042, A4 117.670, A5 -39.183, A6 0.000, E1 3160.09, E2 0, E3 0, E4 0, E5 0, E6 0} C_DIS
   SPTP {A1 5.583, A2 -71.516, A3 89.750, A4 114.197, A5 -36.784, A6 0.000, E1 3166.05, E2 0, E3 0, E4 0, E5 0, E6 0} C_DIS
   SPTP {A1 5.365, A2 -71.925, A3 91.372, A4 110.109, A5 -34.606, A6 0.000, E1 3172.59, E2 0, E3 0, E4 0, E5 0, E6 0} C_DIS
   SPTP {A1 5.159, A2 -72.238, A3 92.906, A4 105.366, A5 -32.694, A6 0.000, E1 3179.74, E2 0, E3 0, E4 0, E5 0, E6 0} C_DIS
   SPTP {A1 4.966, A2 -72.452, A3 94.345, A4 99.967, A5 -31.116, A6 0.000, E1 3187.52, E2 0, E3 0, E4 0, E5 0, E6 0} C_DIS
   SPTP {A1 4.792, A2 -72.549, A3 95.759, A4 93.468, A5 -29.960, A6 0.000, E1 3196.37, E2 0, E3 0, E4 0, E5 0, E6 0} C_DIS
   SPTP {A1 4.626, A2 -72.500, A3 97.176, A4 85.670, A5 -29.383, A6 0.000, E1 3206.45, E2 0, E3 0, E4 0, E5 0, E6 0} C_DIS
   SPTP {A1 4.467, A2 -72.320, A3 98.448, A4 77.717, A5 -29.438, A6 0.000, E1 3216.67, E2 0, E3 0, E4 0, E5 0, E6 0} C_DIS
   SPTP {A1 4.316, A2 -72.011, A3 99.571, A4 69.987, A5 -30.121, A6 0.000, E1 3226.64, E2 0, E3 0, E4 0, E5 0, E6 0} C_DIS
   SPTP {A1 4.174, A2 -71.575, A3 100.540, A4 62.804, A5 -31.383, A6 0.000, E1 3236.06, E2 0, E3 0, E4 0, E5 0, E6 0} C_DIS
   SPTP {A1 4.048, A2 -71.012, A3 101.347, A4 56.397, A5 -33.156, A6 0.000, E1 3244.7, E2 0, E3 0, E4 0, E5 0, E6 0} C_DIS
   SPTP {A1 3.935, A2 -70.330, A3 101.992, A4 50.843, A5 -35.340, A6 0.000, E1 3252.5, E2 0, E3 0, E4 0, E5 0, E6 0} C_DIS
   SPTP {A1 3.837, A2 -69.535, A3 102.473, A4 46.116, A5 -37.841, A6 0.000, E1 3259.49, E2 0, E3 0, E4 0, E5 0, E6 0} C_DIS
   SPTP {A1 3.756, A2 -68.632, A3 102.786, A4 42.165, A5 -40.580, A6 0.000, E1 3265.71, E2 0, E3 0, E4 0, E5 0, E6 0} C_DIS
   SPTP {A1 3.694, A2 -67.629, A3 102.929, A4 38.902, A5 -43.488, A6 0.000, E1 3271.28, E2 0, E3 0, E4 0, E5 0, E6 0} C_DIS
   SPTP {A1 3.644, A2 -66.888, A3 102.987, A4 36.825, A5 -45.637, A6 0.000, E1 3275.38, E2 0, E3 0, E4 0, E5 0, E6 0} C_DIS
   SPTP {A1 3.615, A2 -66.115, A3 102.953, A4 35.102, A5 -47.799, A6 0.000, E1 3279.14, E2 0, E3 0, E4 0, E5 0, E6 0} C_DIS
   SPTP {A1 3.604, A2 -65.298, A3 102.828, A4 33.663, A5 -49.993, A6 0.000, E1 3282.65, E2 0, E3 0, E4 0, E5 0, E6 0} C_DIS
   SPTP {A1 3.612, A2 -64.441, A3 102.611, A4 32.479, A5 -52.202, A6 0.000, E1 3285.93, E2 0, E3 0, E4 0, E5 0, E6 0} C_DIS
   SPTP {A1 3.641, A2 -63.548, A3 102.303, A4 31.532, A5 -54.414, A6 0.000, E1 3289.02, E2 0, E3 0, E4 0, E5 0, E6 0} C_DIS
   SPTP {A1 3.688, A2 -62.621, A3 101.904, A4 30.796, A5 -56.615, A6 0.000, E1 3291.93, E2 0, E3 0, E4 0, E5 0, E6 0} C_DIS
   SPTP {A1 3.773, A2 -61.863, A3 101.517, A4 30.443, A5 -58.378, A6 0.000, E1 3294.48, E2 0, E3 0, E4 0, E5 0, E6 0} C_DIS
   SPTP {A1 3.899, A2 -61.357, A3 101.214, A4 30.478, A5 -59.564, A6 0.000, E1 3296.63, E2 0, E3 0, E4 0, E5 0, E6 0} C_DIS
   SPTP {A1 4.044, A2 -60.841, A3 100.869, A4 30.625, A5 -60.740, A6 0.000, E1 3298.71, E2 0, E3 0, E4 0, E5 0, E6 0} C_DIS
   SPTP {A1 4.202, A2 -60.317, A3 100.486, A4 30.866, A5 -61.900, A6 0.000, E1 3300.71, E2 0, E3 0, E4 0, E5 0, E6 0} C_DIS
   SPTP {A1 4.372, A2 -59.786, A3 100.069, A4 31.181, A5 -63.040, A6 0.000, E1 3302.67, E2 0, E3 0, E4 0, E5 0, E6 0} C_DIS
   SPTP {A1 4.552, A2 -59.250, A3 99.615, A4 31.573, A5 -64.160, A6 0.000, E1 3304.57, E2 0, E3 0, E4 0, E5 0, E6 0} C_DIS
   SPTP {A1 4.742, A2 -58.709, A3 99.125, A4 32.033, A5 -65.258, A6 0.000, E1 3306.42, E2 0, E3 0, E4 0, E5 0, E6 0} C_DIS
   SPTP {A1 4.939, A2 -58.163, A3 98.602, A4 32.552, A5 -66.332, A6 0.000, E1 3308.23, E2 0, E3 0, E4 0, E5 0, E6 0} C_DIS
   SPTP {A1 5.185, A2 -57.844, A3 98.190, A4 33.366, A5 -66.945, A6 0.000, E1 3309.81, E2 0, E3 0, E4 0, E5 0, E6 0} C_DIS
   SPTP {A1 5.462, A2 -57.673, A3 97.848, A4 34.381, A5 -67.260, A6 0.000, E1 3311.21, E2 0, E3 0, E4 0, E5 0, E6 0} C_DIS
   SPTP {A1 5.744, A2 -57.499, A3 97.482, A4 35.438, A5 -67.564, A6 0.000, E1 3312.58, E2 0, E3 0, E4 0, E5 0, E6 0} C_DIS
   SPTP {A1 6.027, A2 -57.324, A3 97.094, A4 36.528, A5 -67.856, A6 0.000, E1 3313.91, E2 0, E3 0, E4 0, E5 0, E6 0} C_DIS
   SPTP {A1 6.312, A2 -57.145, A3 96.683, A4 37.650, A5 -68.137, A6 0.000, E1 3315.22, E2 0, E3 0, E4 0, E5 0, E6 0} C_DIS
   SPTP {A1 6.597, A2 -56.964, A3 96.249, A4 38.801, A5 -68.408, A6 0.000, E1 3316.49, E2 0, E3 0, E4 0, E5 0, E6 0} C_DIS
   SPTP {A1 6.881, A2 -56.780, A3 95.793, A4 39.974, A5 -68.669, A6 0.000, E1 3317.74, E2 0, E3 0, E4 0, E5 0, E6 0} C_DIS
   SPTP {A1 7.162, A2 -56.594, A3 95.316, A4 41.166, A5 -68.920, A6 0.000, E1 3318.97, E2 0, E3 0, E4 0, E5 0, E6 0} C_DIS
   SPTP {A1 7.440, A2 -56.406, A3 94.819, A4 42.373, A5 -69.160, A6 0.000, E1 3320.18, E2 0, E3 0, E4 0, E5 0, E6 0} C_DIS
   SPTP {A1 7.714, A2 -56.217, A3 94.304, A4 43.590, A5 -69.390, A6 0.000, E1 3321.37, E2 0, E3 0, E4 0, E5 0, E6 0} C_DIS
   SPTP {A1 7.981, A2 -56.029, A3 93.774, A4 44.811, A5 -69.607, A6 0.000, E1 3322.56, E2 0, E3 0, E4 0, E5 0, E6 0} C_DIS
   SPTP {A1 8.243, A2 -55.841, A3 93.229, A4 46.035, A5 -69.812, A6 0.000, E1 3323.73, E2 0, E3 0, E4 0, E5 0, E6 0} C_DIS
   SPTP {A1 8.508, A2 -55.757, A3 92.745, A4 47.364, A5 -69.833, A6 0.000, E1 3324.73, E2 0, E3 0, E4 0, E5 0, E6 0} C_DIS
   SPTP {A1 8.768, A2 -55.691, A3 92.259, A4 48.716, A5 -69.816, A6 0.000, E1 3325.68, E2 0, E3 0, E4 0, E5 0, E6 0} C_DIS
   SPTP {A1 9.020, A2 -55.623, A3 91.759, A4 50.070, A5 -69.795, A6 0.000, E1 3326.63, E2 0, E3 0, E4 0, E5 0, E6 0} C_DIS
   SPTP {A1 9.263, A2 -55.554, A3 91.245, A4 51.423, A5 -69.769, A6 0.000, E1 3327.56, E2 0, E3 0, E4 0, E5 0, E6 0} C_DIS
   SPTP {A1 9.498, A2 -55.485, A3 90.721, A4 52.772, A5 -69.738, A6 0.000, E1 3328.49, E2 0, E3 0, E4 0, E5 0, E6 0} C_DIS
   SPTP {A1 9.724, A2 -55.417, A3 90.187, A4 54.116, A5 -69.701, A6 0.000, E1 3329.41, E2 0, E3 0, E4 0, E5 0, E6 0} C_DIS
   SPTP {A1 9.939, A2 -55.350, A3 89.646, A4 55.452, A5 -69.658, A6 0.000, E1 3330.32, E2 0, E3 0, E4 0, E5 0, E6 0} C_DIS
   SPTP {A1 10.145, A2 -55.285, A3 89.100, A4 56.778, A5 -69.607, A6 0.000, E1 3331.24, E2 0, E3 0, E4 0, E5 0, E6 0} C_DIS
   SPTP {A1 10.340, A2 -55.224, A3 88.551, A4 58.093, A5 -69.551, A6 0.000, E1 3332.15, E2 0, E3 0, E4 0, E5 0, E6 0} C_DIS
   SPTP {A1 10.525, A2 -55.168, A3 88.002, A4 59.393, A5 -69.483, A6 0.000, E1 3333.07, E2 0, E3 0, E4 0, E5 0, E6 0} C_DIS
   SPTP {A1 10.690, A2 -55.118, A3 87.476, A4 60.636, A5 -69.420, A6 0.000, E1 3333.97, E2 0, E3 0, E4 0, E5 0, E6 0} C_DIS
   SPTP {A1 10.840, A2 -55.075, A3 86.965, A4 61.839, A5 -69.356, A6 0.000, E1 3334.87, E2 0, E3 0, E4 0, E5 0, E6 0} C_DIS
   SPTP {A1 10.958, A2 -55.041, A3 86.519, A4 62.900, A5 -69.323, A6 0.000, E1 3335.73, E2 0, E3 0, E4 0, E5 0, E6 0} C_DIS
   SPTP {A1 11.062, A2 -55.017, A3 86.095, A4 63.917, A5 -69.286, A6 0.000, E1 3336.6, E2 0, E3 0, E4 0, E5 0, E6 0} C_DIS
   SPTP {A1 11.158, A2 -55.002, A3 85.683, A4 64.915, A5 -69.235, A6 0.000, E1 3337.47, E2 0, E3 0, E4 0, E5 0, E6 0} C_DIS
   SPTP {A1 11.245, A2 -54.997, A3 85.285, A4 65.894, A5 -69.167, A6 0.000, E1 3338.36, E2 0, E3 0, E4 0, E5 0, E6 0} C_DIS
   SPTP {A1 11.324, A2 -55.004, A3 84.903, A4 66.854, A5 -69.083, A6 0.000, E1 3339.27, E2 0, E3 0, E4 0, E5 0, E6 0} C_DIS
   SPTP {A1 11.395, A2 -55.023, A3 84.538, A4 67.795, A5 -68.980, A6 0.000, E1 3340.18, E2 0, E3 0, E4 0, E5 0, E6 0} C_DIS
   SPTP {A1 11.458, A2 -55.056, A3 84.192, A4 68.715, A5 -68.858, A6 0.000, E1 3341.12, E2 0, E3 0, E4 0, E5 0, E6 0} C_DIS
   SPTP {A1 11.513, A2 -55.101, A3 83.865, A4 69.615, A5 -68.717, A6 0.000, E1 3342.06, E2 0, E3 0, E4 0, E5 0, E6 0} C_DIS
   SPTP {A1 11.560, A2 -55.162, A3 83.561, A4 70.494, A5 -68.552, A6 0.000, E1 3343.03, E2 0, E3 0, E4 0, E5 0, E6 0} C_DIS
   SPTP {A1 11.598, A2 -55.238, A3 83.280, A4 71.352, A5 -68.365, A6 0.000, E1 3344, E2 0, E3 0, E4 0, E5 0, E6 0} C_DIS
   SPTP {A1 11.629, A2 -55.330, A3 83.025, A4 72.188, A5 -68.153, A6 0.000, E1 3345, E2 0, E3 0, E4 0, E5 0, E6 0} C_DIS
   SPTP {A1 11.651, A2 -55.437, A3 82.794, A4 73.004, A5 -67.917, A6 0.000, E1 3346.01, E2 0, E3 0, E4 0, E5 0, E6 0} C_DIS
   SPTP {A1 11.666, A2 -55.562, A3 82.590, A4 73.799, A5 -67.656, A6 0.000, E1 3347.04, E2 0, E3 0, E4 0, E5 0, E6 0} C_DIS
   SPTP {A1 11.673, A2 -55.703, A3 82.413, A4 74.573, A5 -67.368, A6 0.000, E1 3348.08, E2 0, E3 0, E4 0, E5 0, E6 0} C_DIS
   SPTP {A1 11.672, A2 -55.861, A3 82.265, A4 75.326, A5 -67.052, A6 0.000, E1 3349.14, E2 0, E3 0, E4 0, E5 0, E6 0} C_DIS
   SPTP {A1 11.663, A2 -56.036, A3 82.146, A4 76.057, A5 -66.708, A6 0.000, E1 3350.21, E2 0, E3 0, E4 0, E5 0, E6 0} C_DIS
   SPTP {A1 11.647, A2 -56.229, A3 82.056, A4 76.768, A5 -66.335, A6 0.000, E1 3351.3, E2 0, E3 0, E4 0, E5 0, E6 0} C_DIS
   SPTP {A1 11.616, A2 -56.482, A3 82.043, A4 77.487, A5 -65.907, A6 0.000, E1 3352.16, E2 0, E3 0, E4 0, E5 0, E6 0} C_DIS
   SPTP {A1 11.576, A2 -56.759, A3 82.065, A4 78.199, A5 -65.447, A6 0.000, E1 3352.95, E2 0, E3 0, E4 0, E5 0, E6 0} C_DIS
   SPTP {A1 11.529, A2 -57.047, A3 82.106, A4 78.898, A5 -64.967, A6 0.000, E1 3353.75, E2 0, E3 0, E4 0, E5 0, E6 0} C_DIS
   SPTP {A1 11.475, A2 -57.348, A3 82.169, A4 79.584, A5 -64.462, A6 0.000, E1 3354.55, E2 0, E3 0, E4 0, E5 0, E6 0} C_DIS
   SPTP {A1 11.413, A2 -57.661, A3 82.252, A4 80.256, A5 -63.933, A6 0.000, E1 3355.37, E2 0, E3 0, E4 0, E5 0, E6 0} C_DIS
   SPTP {A1 11.344, A2 -57.987, A3 82.357, A4 80.913, A5 -63.377, A6 0.000, E1 3356.18, E2 0, E3 0, E4 0, E5 0, E6 0} C_DIS
   SPTP {A1 11.267, A2 -58.326, A3 82.484, A4 81.555, A5 -62.794, A6 0.000, E1 3357.01, E2 0, E3 0, E4 0, E5 0, E6 0} C_DIS
   SPTP {A1 11.183, A2 -58.677, A3 82.633, A4 82.183, A5 -62.184, A6 0.000, E1 3357.84, E2 0, E3 0, E4 0, E5 0, E6 0} C_DIS
   SPTP {A1 11.090, A2 -59.041, A3 82.802, A4 82.798, A5 -61.546, A6 0.000, E1 3358.67, E2 0, E3 0, E4 0, E5 0, E6 0} C_DIS
   SPTP {A1 10.989, A2 -59.415, A3 82.992, A4 83.398, A5 -60.881, A6 0.000, E1 3359.51, E2 0, E3 0, E4 0, E5 0, E6 0} C_DIS
   SPTP {A1 10.880, A2 -59.801, A3 83.203, A4 83.984, A5 -60.187, A6 0.000, E1 3360.36, E2 0, E3 0, E4 0, E5 0, E6 0} C_DIS
   SPTP {A1 10.762, A2 -60.198, A3 83.432, A4 84.557, A5 -59.464, A6 0.000, E1 3361.2, E2 0, E3 0, E4 0, E5 0, E6 0} C_DIS
   SPTP {A1 10.643, A2 -60.663, A3 83.579, A4 85.600, A5 -58.594, A6 0.000, E1 3361.5, E2 0, E3 0, E4 0, E5 0, E6 0} C_DIS
   SPTP {A1 10.513, A2 -61.137, A3 83.718, A4 86.703, A5 -57.700, A6 0.000, E1 3361.73, E2 0, E3 0, E4 0, E5 0, E6 0} C_DIS
   SPTP {A1 10.373, A2 -61.613, A3 83.864, A4 87.820, A5 -56.789, A6 0.000, E1 3361.92, E2 0, E3 0, E4 0, E5 0, E6 0} C_DIS
   SPTP {A1 10.220, A2 -62.090, A3 84.015, A4 88.950, A5 -55.866, A6 0.000, E1 3362.09, E2 0, E3 0, E4 0, E5 0, E6 0} C_DIS
   SPTP {A1 10.056, A2 -62.568, A3 84.170, A4 90.096, A5 -54.931, A6 0.000, E1 3362.23, E2 0, E3 0, E4 0, E5 0, E6 0} C_DIS
   SPTP {A1 9.880, A2 -63.045, A3 84.328, A4 91.262, A5 -53.986, A6 0.000, E1 3362.35, E2 0, E3 0, E4 0, E5 0, E6 0} C_DIS
   SPTP {A1 9.693, A2 -63.522, A3 84.490, A4 92.447, A5 -53.030, A6 0.000, E1 3362.42, E2 0, E3 0, E4 0, E5 0, E6 0} C_DIS
   SPTP {A1 9.494, A2 -63.998, A3 84.654, A4 93.655, A5 -52.062, A6 0.000, E1 3362.47, E2 0, E3 0, E4 0, E5 0, E6 0} C_DIS
   SPTP {A1 9.283, A2 -64.473, A3 84.822, A4 94.887, A5 -51.085, A6 0.000, E1 3362.47, E2 0, E3 0, E4 0, E5 0, E6 0} C_DIS
   SPTP {A1 9.060, A2 -64.946, A3 84.992, A4 96.148, A5 -50.098, A6 0.000, E1 3362.44, E2 0, E3 0, E4 0, E5 0, E6 0} C_DIS
   SPTP {A1 8.824, A2 -65.417, A3 85.164, A4 97.439, A5 -49.102, A6 0.000, E1 3362.36, E2 0, E3 0, E4 0, E5 0, E6 0} C_DIS
   SPTP {A1 8.576, A2 -65.885, A3 85.338, A4 98.763, A5 -48.099, A6 0.000, E1 3362.24, E2 0, E3 0, E4 0, E5 0, E6 0} C_DIS
   SPTP {A1 8.316, A2 -66.349, A3 85.513, A4 100.125, A5 -47.091, A6 0.000, E1 3362.07, E2 0, E3 0, E4 0, E5 0, E6 0} C_DIS
   SPTP {A1 8.045, A2 -66.809, A3 85.686, A4 101.530, A5 -46.080, A6 0.000, E1 3361.85, E2 0, E3 0, E4 0, E5 0, E6 0} C_DIS
   SPTP {A1 7.762, A2 -67.262, A3 85.845, A4 103.029, A5 -45.066, A6 0.000, E1 3361.55, E2 0, E3 0, E4 0, E5 0, E6 0} C_DIS
   SPTP {A1 7.450, A2 -67.720, A3 85.907, A4 105.006, A5 -43.979, A6 0.000, E1 3360.96, E2 0, E3 0, E4 0, E5 0, E6 0} C_DIS
   SPTP {A1 7.125, A2 -68.167, A3 85.964, A4 107.060, A5 -42.914, A6 0.000, E1 3360.29, E2 0, E3 0, E4 0, E5 0, E6 0} C_DIS
   SPTP {A1 6.785, A2 -68.603, A3 86.019, A4 109.195, A5 -41.868, A6 0.000, E1 3359.52, E2 0, E3 0, E4 0, E5 0, E6 0} C_DIS
   SPTP {A1 6.431, A2 -69.027, A3 86.070, A4 111.414, A5 -40.846, A6 0.000, E1 3358.67, E2 0, E3 0, E4 0, E5 0, E6 0} C_DIS
   SPTP {A1 6.063, A2 -69.440, A3 86.118, A4 113.724, A5 -39.850, A6 0.000, E1 3357.72, E2 0, E3 0, E4 0, E5 0, E6 0} C_DIS
   SPTP {A1 5.682, A2 -69.839, A3 86.161, A4 116.127, A5 -38.889, A6 0.000, E1 3356.67, E2 0, E3 0, E4 0, E5 0, E6 0} C_DIS
   SPTP {A1 5.290, A2 -70.223, A3 86.198, A4 118.626, A5 -37.971, A6 0.000, E1 3355.52, E2 0, E3 0, E4 0, E5 0, E6 0} C_DIS
   SPTP {A1 4.889, A2 -70.592, A3 86.228, A4 121.220, A5 -37.102, A6 0.000, E1 3354.28, E2 0, E3 0, E4 0, E5 0, E6 0} C_DIS
   SPTP {A1 4.478, A2 -70.944, A3 86.252, A4 123.909, A5 -36.289, A6 0.000, E1 3352.95, E2 0, E3 0, E4 0, E5 0, E6 0} C_DIS
   SPTP {A1 4.060, A2 -71.279, A3 86.268, A4 126.688, A5 -35.537, A6 0.000, E1 3351.52, E2 0, E3 0, E4 0, E5 0, E6 0} C_DIS
   SPTP {A1 3.635, A2 -71.599, A3 86.279, A4 129.552, A5 -34.848, A6 0.000, E1 3350.02, E2 0, E3 0, E4 0, E5 0, E6 0} C_DIS
   SPTP {A1 3.204, A2 -71.903, A3 86.286, A4 132.496, A5 -34.222, A6 0.000, E1 3348.45, E2 0, E3 0, E4 0, E5 0, E6 0} C_DIS
   SPTP {A1 2.770, A2 -72.190, A3 86.286, A4 135.502, A5 -33.675, A6 0.000, E1 3346.82, E2 0, E3 0, E4 0, E5 0, E6 0} C_DIS
   SPTP {A1 2.336, A2 -72.508, A3 86.467, A4 138.161, A5 -32.912, A6 0.000, E1 3345.64, E2 0, E3 0, E4 0, E5 0, E6 0} C_DIS
   SPTP {A1 1.900, A2 -72.884, A3 86.912, A4 140.344, A5 -31.771, A6 0.000, E1 3345.07, E2 0, E3 0, E4 0, E5 0, E6 0} C_DIS
   SPTP {A1 1.467, A2 -73.248, A3 87.364, A4 142.606, A5 -30.654, A6 0.000, E1 3344.42, E2 0, E3 0, E4 0, E5 0, E6 0} C_DIS
   SPTP {A1 1.036, A2 -73.601, A3 87.822, A4 144.957, A5 -29.559, A6 0.000, E1 3343.68, E2 0, E3 0, E4 0, E5 0, E6 0} C_DIS
   SPTP {A1 0.615, A2 -73.941, A3 88.286, A4 147.370, A5 -28.500, A6 0.000, E1 3342.9, E2 0, E3 0, E4 0, E5 0, E6 0} C_DIS
   SPTP {A1 0.207, A2 -74.269, A3 88.755, A4 149.834, A5 -27.480, A6 0.000, E1 3342.08, E2 0, E3 0, E4 0, E5 0, E6 0} C_DIS
   SPTP {A1 -0.184, A2 -74.586, A3 89.231, A4 152.325, A5 -26.500, A6 0.000, E1 3341.26, E2 0, E3 0, E4 0, E5 0, E6 0} C_DIS
   SPTP {A1 -0.552, A2 -74.919, A3 89.829, A4 154.563, A5 -25.344, A6 0.000, E1 3340.71, E2 0, E3 0, E4 0, E5 0, E6 0} C_DIS
   SPTP {A1 -0.885, A2 -75.365, A3 91.023, A4 155.437, A5 -23.081, A6 0.000, E1 3341.54, E2 0, E3 0, E4 0, E5 0, E6 0} C_DIS
   SPTP {A1 -1.191, A2 -75.776, A3 92.200, A4 156.210, A5 -20.819, A6 0.000, E1 3342.47, E2 0, E3 0, E4 0, E5 0, E6 0} C_DIS
   SPTP {A1 -1.461, A2 -76.152, A3 93.357, A4 156.787, A5 -18.567, A6 0.000, E1 3343.62, E2 0, E3 0, E4 0, E5 0, E6 0} C_DIS
   SPTP {A1 -1.690, A2 -76.492, A3 94.495, A4 157.044, A5 -16.328, A6 0.000, E1 3345.12, E2 0, E3 0, E4 0, E5 0, E6 0} C_DIS
   SPTP {A1 -1.871, A2 -76.806, A3 95.718, A4 156.305, A5 -13.872, A6 0.000, E1 3347.63, E2 0, E3 0, E4 0, E5 0, E6 0} C_DIS
   SPTP {A1 -2.003, A2 -77.094, A3 97.560, A4 149.942, A5 -9.948, A6 0.000, E1 3355.72, E2 0, E3 0, E4 0, E5 0, E6 0} C_DIS
   SPTP {A1 -2.084, A2 -77.257, A3 99.287, A4 134.526, A5 -6.397, A6 0.000, E1 3372.87, E2 0, E3 0, E4 0, E5 0, E6 0} C_DIS
   SPTP {A1 -2.113, A2 -77.292, A3 100.892, A4 94.451, A5 -4.328, A6 0.000, E1 3414.68, E2 0, E3 0, E4 0, E5 0, E6 0} C_DIS
   SPTP {A1 -2.086, A2 -77.196, A3 102.370, A4 48.000, A5 -5.727, A6 0.000, E1 3462.89, E2 0, E3 0, E4 0, E5 0, E6 0} C_DIS
   SPTP {A1 -2.021, A2 -76.795, A3 104.074, A4 24.670, A5 -10.441, A6 0.000, E1 3488, E2 0, E3 0, E4 0, E5 0, E6 0} C_DIS
   SPTP {A1 -1.911, A2 -76.029, A3 105.670, A4 16.308, A5 -16.585, A6 0.000, E1 3498.15, E2 0, E3 0, E4 0, E5 0, E6 0} C_DIS
   SPTP {A1 -1.765, A2 -74.973, A3 106.918, A4 12.944, A5 -22.879, A6 0.000, E1 3503.29, E2 0, E3 0, E4 0, E5 0, E6 0} C_DIS
   SPTP {A1 -1.599, A2 -73.517, A3 107.843, A4 11.130, A5 -29.626, A6 0.000, E1 3506.95, E2 0, E3 0, E4 0, E5 0, E6 0} C_DIS
   SPTP {A1 -1.410, A2 -71.237, A3 108.342, A4 9.789, A5 -37.925, A6 0.000, E1 3510.38, E2 0, E3 0, E4 0, E5 0, E6 0} C_DIS
   SPTP {A1 -1.212, A2 -68.564, A3 108.158, A4 9.179, A5 -45.975, A6 0.000, E1 3513.1, E2 0, E3 0, E4 0, E5 0, E6 0} C_DIS
   SPTP {A1 -1.013, A2 -65.570, A3 107.290, A4 8.963, A5 -53.683, A6 0.000, E1 3515.45, E2 0, E3 0, E4 0, E5 0, E6 0} C_DIS
   SPTP {A1 -0.809, A2 -62.400, A3 105.787, A4 8.999, A5 -60.828, A6 0.000, E1 3517.67, E2 0, E3 0, E4 0, E5 0, E6 0} C_DIS
   SPTP {A1 -0.388, A2 -59.786, A3 104.136, A4 9.840, A5 -66.146, A6 0.000, E1 3519.98, E2 0, E3 0, E4 0, E5 0, E6 0} C_DIS
   SPTP {A1 0.049, A2 -57.114, A3 102.092, A4 10.818, A5 -71.109, A6 0.000, E1 3522.25, E2 0, E3 0, E4 0, E5 0, E6 0} C_DIS
   SPTP {A1 0.502, A2 -54.409, A3 99.672, A4 11.946, A5 -75.706, A6 0.000, E1 3524.49, E2 0, E3 0, E4 0, E5 0, E6 0} C_DIS
   SPTP {A1 0.965, A2 -51.695, A3 96.893, A4 13.200, A5 -79.928, A6 0.000, E1 3526.7, E2 0, E3 0, E4 0, E5 0, E6 0} C_DIS
   SPTP {A1 1.432, A2 -48.985, A3 93.772, A4 14.569, A5 -83.772, A6 0.000, E1 3528.89, E2 0, E3 0, E4 0, E5 0, E6 0} C_DIS
   SPTP {A1 1.902, A2 -46.286, A3 90.318, A4 16.053, A5 -87.245, A6 0.000, E1 3531.05, E2 0, E3 0, E4 0, E5 0, E6 0} C_DIS
   SPTP {A1 2.376, A2 -43.590, A3 86.529, A4 17.666, A5 -90.358, A6 0.000, E1 3533.16, E2 0, E3 0, E4 0, E5 0, E6 0} C_DIS
   SPTP {A1 2.847, A2 -40.892, A3 82.401, A4 19.385, A5 -93.117, A6 0.000, E1 3535.2, E2 0, E3 0, E4 0, E5 0, E6 0} C_DIS
   SPTP {A1 3.313, A2 -38.170, A3 77.914, A4 21.200, A5 -95.532, A6 0.000, E1 3537.16, E2 0, E3 0, E4 0, E5 0, E6 0} C_DIS
   SPTP {A1 3.770, A2 -35.395, A3 73.027, A4 23.102, A5 -97.606, A6 0.000, E1 3539, E2 0, E3 0, E4 0, E5 0, E6 0} C_DIS
   SPTP {A1 4.316, A2 -34.784, A3 71.505, A4 25.234, A5 -97.894, A6 0.000, E1 3540.36, E2 0, E3 0, E4 0, E5 0, E6 0} C_DIS
   SPTP {A1 4.878, A2 -34.655, A3 70.719, A4 27.472, A5 -97.793, A6 0.000, E1 3541.49, E2 0, E3 0, E4 0, E5 0, E6 0} C_DIS
   SPTP {A1 5.429, A2 -34.500, A3 69.837, A4 29.764, A5 -97.664, A6 0.000, E1 3542.46, E2 0, E3 0, E4 0, E5 0, E6 0} C_DIS
   SPTP {A1 5.960, A2 -34.443, A3 69.083, A4 32.059, A5 -97.441, A6 0.000, E1 3543.26, E2 0, E3 0, E4 0, E5 0, E6 0} C_DIS
   SPTP {A1 6.439, A2 -35.085, A3 69.533, A4 34.194, A5 -96.774, A6 0.000, E1 3543.64, E2 0, E3 0, E4 0, E5 0, E6 0} C_DIS
   SPTP {A1 6.909, A2 -35.679, A3 69.857, A4 36.364, A5 -96.096, A6 0.000, E1 3543.9, E2 0, E3 0, E4 0, E5 0, E6 0} C_DIS
   SPTP {A1 7.177, A2 -36.003, A3 69.993, A4 37.629, A5 -95.702, A6 0.000, E1 3544, E2 0, E3 0, E4 0, E5 0, E6 0} C_DIS
   SPTP {A1 7.441, A2 -36.315, A3 70.093, A4 38.902, A5 -95.305, A6 0.000, E1 3544.07, E2 0, E3 0, E4 0, E5 0, E6 0} C_DIS
   SPTP {A1 7.442, A2 -36.300, A3 70.075, A4 38.915, A5 -95.317, A6 0.000, E1 3544.05, E2 0, E3 0, E4 0, E5 0, E6 0} C_DIS
   SPTP {A1 7.889, A2 -36.813, A3 70.178, A4 41.122, A5 -94.628, A6 0.000, E1 3544.12, E2 0, E3 0, E4 0, E5 0, E6 0} C_DIS
   SPTP {A1 8.293, A2 -37.569, A3 70.695, A4 43.198, A5 -93.772, A6 0.000, E1 3543.95, E2 0, E3 0, E4 0, E5 0, E6 0} C_DIS
   SPTP {A1 8.658, A2 -38.569, A3 71.619, A4 45.155, A5 -92.732, A6 0.000, E1 3543.5, E2 0, E3 0, E4 0, E5 0, E6 0} C_DIS
   SPTP {A1 9.014, A2 -39.541, A3 72.448, A4 47.120, A5 -91.667, A6 0.000, E1 3543, E2 0, E3 0, E4 0, E5 0, E6 0} C_DIS
   SPTP {A1 9.363, A2 -40.483, A3 73.179, A4 49.105, A5 -90.587, A6 0.000, E1 3542.43, E2 0, E3 0, E4 0, E5 0, E6 0} C_DIS
   SPTP {A1 9.701, A2 -41.400, A3 73.826, A4 51.100, A5 -89.494, A6 0.000, E1 3541.8, E2 0, E3 0, E4 0, E5 0, E6 0} C_DIS
   SPTP {A1 10.027, A2 -42.300, A3 74.403, A4 53.102, A5 -88.385, A6 0.000, E1 3541.13, E2 0, E3 0, E4 0, E5 0, E6 0} C_DIS
   SPTP {A1 10.340, A2 -43.189, A3 74.926, A4 55.105, A5 -87.257, A6 0.000, E1 3540.43, E2 0, E3 0, E4 0, E5 0, E6 0} C_DIS
   SPTP {A1 10.636, A2 -44.069, A3 75.397, A4 57.108, A5 -86.113, A6 0.000, E1 3539.68, E2 0, E3 0, E4 0, E5 0, E6 0} C_DIS
   SPTP {A1 10.895, A2 -45.049, A3 76.026, A4 59.019, A5 -84.888, A6 0.000, E1 3538.72, E2 0, E3 0, E4 0, E5 0, E6 0} C_DIS
   SPTP {A1 11.127, A2 -46.072, A3 76.696, A4 60.894, A5 -83.609, A6 0.000, E1 3537.63, E2 0, E3 0, E4 0, E5 0, E6 0} C_DIS
   SPTP {A1 11.345, A2 -47.063, A3 77.276, A4 62.807, A5 -82.339, A6 0.000, E1 3536.47, E2 0, E3 0, E4 0, E5 0, E6 0} C_DIS
   SPTP {A1 11.545, A2 -48.051, A3 77.813, A4 64.729, A5 -81.048, A6 0.000, E1 3535.25, E2 0, E3 0, E4 0, E5 0, E6 0} C_DIS
   SPTP {A1 11.727, A2 -49.019, A3 78.284, A4 66.681, A5 -79.760, A6 0.000, E1 3533.96, E2 0, E3 0, E4 0, E5 0, E6 0} C_DIS
   SPTP {A1 11.887, A2 -49.982, A3 78.712, A4 68.649, A5 -78.459, A6 0.000, E1 3532.61, E2 0, E3 0, E4 0, E5 0, E6 0} C_DIS
   SPTP {A1 12.026, A2 -50.929, A3 79.085, A4 70.647, A5 -77.162, A6 0.000, E1 3531.19, E2 0, E3 0, E4 0, E5 0, E6 0} C_DIS
   SPTP {A1 12.143, A2 -51.859, A3 79.402, A4 72.680, A5 -75.872, A6 0.000, E1 3529.7, E2 0, E3 0, E4 0, E5 0, E6 0} C_DIS
   SPTP {A1 12.235, A2 -52.775, A3 79.672, A4 74.746, A5 -74.589, A6 0.000, E1 3528.13, E2 0, E3 0, E4 0, E5 0, E6 0} C_DIS
   SPTP {A1 12.304, A2 -53.666, A3 79.877, A4 76.862, A5 -73.333, A6 0.000, E1 3526.47, E2 0, E3 0, E4 0, E5 0, E6 0} C_DIS
   SPTP {A1 12.347, A2 -54.542, A3 80.038, A4 79.016, A5 -72.090, A6 0.000, E1 3524.72, E2 0, E3 0, E4 0, E5 0, E6 0} C_DIS
   SPTP {A1 12.365, A2 -55.383, A3 80.125, A4 81.234, A5 -70.896, A6 0.000, E1 3522.88, E2 0, E3 0, E4 0, E5 0, E6 0} C_DIS
   SPTP {A1 12.354, A2 -56.207, A3 80.168, A4 83.499, A5 -69.726, A6 0.000, E1 3520.94, E2 0, E3 0, E4 0, E5 0, E6 0} C_DIS
   SPTP {A1 12.317, A2 -56.979, A3 80.139, A4 85.792, A5 -68.633, A6 0.000, E1 3518.98, E2 0, E3 0, E4 0, E5 0, E6 0} C_DIS
   SPTP {A1 12.250, A2 -57.668, A3 80.101, A4 87.867, A5 -67.620, A6 0.000, E1 3517.48, E2 0, E3 0, E4 0, E5 0, E6 0} C_DIS
   SPTP {A1 12.158, A2 -58.333, A3 80.033, A4 89.960, A5 -66.644, A6 0.000, E1 3515.97, E2 0, E3 0, E4 0, E5 0, E6 0} C_DIS
   SPTP {A1 12.043, A2 -58.979, A3 79.935, A4 92.099, A5 -65.699, A6 0.000, E1 3514.38, E2 0, E3 0, E4 0, E5 0, E6 0} C_DIS
   SPTP {A1 11.903, A2 -59.604, A3 79.802, A4 94.289, A5 -64.795, A6 0.000, E1 3512.72, E2 0, E3 0, E4 0, E5 0, E6 0} C_DIS
   SPTP {A1 11.740, A2 -60.202, A3 79.629, A4 96.533, A5 -63.943, A6 0.000, E1 3510.97, E2 0, E3 0, E4 0, E5 0, E6 0} C_DIS
   SPTP {A1 11.553, A2 -60.773, A3 79.416, A4 98.833, A5 -63.147, A6 0.000, E1 3509.15, E2 0, E3 0, E4 0, E5 0, E6 0} C_DIS
   SPTP {A1 11.345, A2 -61.307, A3 79.149, A4 101.193, A5 -62.431, A6 0.000, E1 3507.25, E2 0, E3 0, E4 0, E5 0, E6 0} C_DIS
   SPTP {A1 11.117, A2 -61.799, A3 78.836, A4 103.586, A5 -61.796, A6 0.000, E1 3505.32, E2 0, E3 0, E4 0, E5 0, E6 0} C_DIS
   SPTP {A1 10.872, A2 -62.301, A3 78.792, A4 105.415, A5 -60.982, A6 0.000, E1 3504.5, E2 0, E3 0, E4 0, E5 0, E6 0} C_DIS
   SPTP {A1 10.610, A2 -62.792, A3 78.738, A4 107.284, A5 -60.191, A6 0.000, E1 3503.63, E2 0, E3 0, E4 0, E5 0, E6 0} C_DIS
   SPTP {A1 10.331, A2 -63.267, A3 78.672, A4 109.194, A5 -59.429, A6 0.000, E1 3502.71, E2 0, E3 0, E4 0, E5 0, E6 0} C_DIS
   SPTP {A1 10.039, A2 -63.720, A3 78.583, A4 111.149, A5 -58.715, A6 0.000, E1 3501.74, E2 0, E3 0, E4 0, E5 0, E6 0} C_DIS
   SPTP {A1 9.735, A2 -64.145, A3 78.464, A4 113.147, A5 -58.062, A6 0.000, E1 3500.72, E2 0, E3 0, E4 0, E5 0, E6 0} C_DIS
   SPTP {A1 9.423, A2 -64.539, A3 78.311, A4 115.188, A5 -57.483, A6 0.000, E1 3499.67, E2 0, E3 0, E4 0, E5 0, E6 0} C_DIS
   SPTP {A1 9.105, A2 -64.981, A3 78.402, A4 116.844, A5 -56.689, A6 0.000, E1 3499.3, E2 0, E3 0, E4 0, E5 0, E6 0} C_DIS
   SPTP {A1 8.783, A2 -65.506, A3 78.828, A4 118.011, A5 -55.558, A6 0.000, E1 3499.74, E2 0, E3 0, E4 0, E5 0, E6 0} C_DIS
   SPTP {A1 8.458, A2 -66.016, A3 79.248, A4 119.192, A5 -54.443, A6 0.000, E1 3500.17, E2 0, E3 0, E4 0, E5 0, E6 0} C_DIS
   SPTP {A1 8.132, A2 -66.509, A3 79.661, A4 120.385, A5 -53.352, A6 0.000, E1 3500.6, E2 0, E3 0, E4 0, E5 0, E6 0} C_DIS
   SPTP {A1 7.809, A2 -66.980, A3 80.061, A4 121.586, A5 -52.294, A6 0.000, E1 3501.03, E2 0, E3 0, E4 0, E5 0, E6 0} C_DIS
   SPTP {A1 7.491, A2 -67.450, A3 80.514, A4 122.685, A5 -51.198, A6 0.000, E1 3501.63, E2 0, E3 0, E4 0, E5 0, E6 0} C_DIS
   SPTP {A1 7.185, A2 -68.105, A3 81.681, A4 122.553, A5 -49.291, A6 0.000, E1 3503.95, E2 0, E3 0, E4 0, E5 0, E6 0} C_DIS
   SPTP {A1 6.886, A2 -68.729, A3 82.834, A4 122.312, A5 -47.393, A6 0.000, E1 3506.37, E2 0, E3 0, E4 0, E5 0, E6 0} C_DIS
   SPTP {A1 6.597, A2 -69.318, A3 83.967, A4 121.948, A5 -45.517, A6 0.000, E1 3508.9, E2 0, E3 0, E4 0, E5 0, E6 0} C_DIS
   SPTP {A1 6.318, A2 -69.873, A3 85.079, A4 121.446, A5 -43.668, A6 0.000, E1 3511.55, E2 0, E3 0, E4 0, E5 0, E6 0} C_DIS
   SPTP {A1 6.054, A2 -70.403, A3 86.229, A4 120.632, A5 -41.786, A6 0.000, E1 3514.55, E2 0, E3 0, E4 0, E5 0, E6 0} C_DIS
   SPTP {A1 5.810, A2 -71.006, A3 88.023, A4 117.732, A5 -39.204, A6 0.000, E1 3519.97, E2 0, E3 0, E4 0, E5 0, E6 0} C_DIS
   SPTP {A1 5.579, A2 -71.513, A3 89.732, A4 114.274, A5 -36.801, A6 0.000, E1 3525.91, E2 0, E3 0, E4 0, E5 0, E6 0} C_DIS
   SPTP {A1 5.360, A2 -71.925, A3 91.354, A4 110.201, A5 -34.616, A6 0.000, E1 3532.42, E2 0, E3 0, E4 0, E5 0, E6 0} C_DIS
   SPTP {A1 5.153, A2 -72.240, A3 92.889, A4 105.475, A5 -32.696, A6 0.000, E1 3539.56, E2 0, E3 0, E4 0, E5 0, E6 0} C_DIS
   SPTP {A1 4.959, A2 -72.457, A3 94.328, A4 100.092, A5 -31.107, A6 0.000, E1 3547.32, E2 0, E3 0, E4 0, E5 0, E6 0} C_DIS
   SPTP {A1 4.784, A2 -72.557, A3 95.738, A4 93.641, A5 -29.940, A6 0.000, E1 3556.12, E2 0, E3 0, E4 0, E5 0, E6 0} C_DIS
   SPTP {A1 4.618, A2 -72.511, A3 97.156, A4 85.851, A5 -29.347, A6 0.000, E1 3566.19, E2 0, E3 0, E4 0, E5 0, E6 0} C_DIS
   SPTP {A1 4.458, A2 -72.335, A3 98.431, A4 77.894, A5 -29.385, A6 0.000, E1 3576.41, E2 0, E3 0, E4 0, E5 0, E6 0} C_DIS
   SPTP {A1 4.307, A2 -72.030, A3 99.557, A4 70.152, A5 -30.050, A6 0.000, E1 3586.39, E2 0, E3 0, E4 0, E5 0, E6 0} C_DIS
   SPTP {A1 4.165, A2 -71.598, A3 100.529, A4 62.951, A5 -31.297, A6 0.000, E1 3595.82, E2 0, E3 0, E4 0, E5 0, E6 0} C_DIS
   SPTP {A1 4.038, A2 -71.040, A3 101.340, A4 56.523, A5 -33.057, A6 0.000, E1 3604.49, E2 0, E3 0, E4 0, E5 0, E6 0} C_DIS
   SPTP {A1 3.926, A2 -70.363, A3 101.989, A4 50.946, A5 -35.230, A6 0.000, E1 3612.31, E2 0, E3 0, E4 0, E5 0, E6 0} C_DIS
   SPTP {A1 3.827, A2 -69.572, A3 102.474, A4 46.202, A5 -37.722, A6 0.000, E1 3619.3, E2 0, E3 0, E4 0, E5 0, E6 0} C_DIS
   SPTP {A1 3.747, A2 -68.674, A3 102.792, A4 42.234, A5 -40.453, A6 0.000, E1 3625.54, E2 0, E3 0, E4 0, E5 0, E6 0} C_DIS
   SPTP {A1 3.685, A2 -67.675, A3 102.942, A4 38.956, A5 -43.356, A6 0.000, E1 3631.12, E2 0, E3 0, E4 0, E5 0, E6 0} C_DIS
   SPTP {A1 3.635, A2 -66.922, A3 103.001, A4 36.843, A5 -45.537, A6 0.000, E1 3635.27, E2 0, E3 0, E4 0, E5 0, E6 0} C_DIS
   SPTP {A1 3.606, A2 -66.151, A3 102.970, A4 35.115, A5 -47.698, A6 0.000, E1 3639.03, E2 0, E3 0, E4 0, E5 0, E6 0} C_DIS
   SPTP {A1 3.595, A2 -65.336, A3 102.848, A4 33.671, A5 -49.890, A6 0.000, E1 3642.54, E2 0, E3 0, E4 0, E5 0, E6 0} C_DIS
   SPTP {A1 3.603, A2 -64.482, A3 102.635, A4 32.482, A5 -52.098, A6 0.000, E1 3645.83, E2 0, E3 0, E4 0, E5 0, E6 0} C_DIS
   SPTP {A1 3.632, A2 -63.590, A3 102.329, A4 31.533, A5 -54.310, A6 0.000, E1 3648.91, E2 0, E3 0, E4 0, E5 0, E6 0} C_DIS

   $VEL.CP=0.167
   HALT
   ;GO_HOME()
   PTP {A1 -30.000, A2 -120.000, A3 120.000, A4 0.000, A5 0.000, A6 0.000, E1 0, E2 0, E3 0, E4 0, E5 0, E6 0}
   ;ENDIF
   $async_EX_AX_DECOUPLE='b0001' ;dianji qu ouhe
   $AXIS_ACT.E1=0 ;bianmqi qingling
   WAIT SEC 1 ; yanshi 1s
   $async_EX_AX_DECOUPLE='b0000' ;dianji ouhe
END
